FUNCTION_BLOCK BaseModuleToBeVisited IMPLEMENTS ITF_Base
VAR
	_name : STRING;
	_hasError : BOOL;
	_errorMessage : STRING;
END_VAR

METHOD Accept : BOOL
VAR_INPUT
	Visitor : ITF_Visitor;
END_VAR
Visitor.VisitBaseObject(this^);
END_METHOD

METHOD FB_init : BOOL
VAR_INPUT
	bInitRetains : BOOL; // if TRUE, the retain variables are initialized (warm start / cold start)
	bInCopyCode : BOOL;  // if TRUE, the instance afterwards gets moved into the copy code (online change)
	MyName : STRING;
END_VAR
_name := MyName;
END_METHOD

METHOD GetErrorMessage : STRING
GetErrorMessage := _errorMessage;
END_METHOD

METHOD HasError : BOOL
HasError := _hasError;
END_METHOD

PROPERTY Name : STRING
GET
Name := _name;
END_GET
END_PROPERTY

END_FUNCTION_BLOCK

(* stored: Version 1.1.0.1, ProductVersion 3.1.4024.12
   POU BaseModuleToBeVisited: Id {9c224321-3b67-448a-a299-36162a20404a}, SpecialFunc None
   Method Accept: Id {0acaeaba-b5f6-4c03-a296-6f390c6c03c9}
   Method FB_init: Id {f9b3a16f-2d92-4a5d-91a6-71636c4aa458}
   Method GetErrorMessage: Id {70271b55-1684-4672-aa47-71665e5e3716}
   Method HasError: Id {357c5fcb-ca55-45b3-b298-56d969f38857}
   Property Name: Id {02d61ea3-f993-4099-9cfe-d42c0891d2e9}
   Get Get: Id {8d44a1f0-d5f7-47a7-8d7e-57d1008d888b} *)
